FUNCTION_BLOCK SS4_ifb_Laser_1 (* Basic FB with empty ECC *)
  (* Standard: 61499-2 *)
  (* Version 1.0, 2021-08-23, AK121668 *)
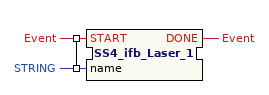
  EVENT_INPUT
    START WITH name;
  END_EVENT
  EVENT_OUTPUT
    DONE;
  END_EVENT
  VAR_INPUT
    name : STRING := 'Well Done!';
  END_VAR
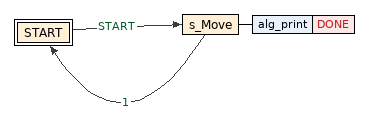
  EC_STATES
    START; (* Initial State *)
    s_Move : alg_print -> DONE;
  END_STATES
  EC_TRANSITIONS
    START TO s_Move := START;
    s_Move TO START := 1;
  END_TRANSITIONS
  ALGORITHM alg_init IN ST:

  END_ALGORITHM
  ALGORITHM alg_print IN ST:

  END_ALGORITHM
  ALGORITHM alg_print_Done IN ST:

  END_ALGORITHM
END_FUNCTION_BLOCK
